PROGRAM Fast
VAR
	SerialLineControl1:SerialLineControl;
END_VAR

//编码器任务周期
serial1fast();

ACTION Serial1Fast:
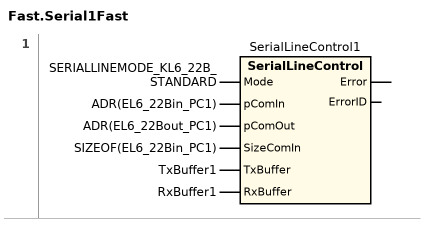
// NETWORK 1
SerialLineControl1(
    Mode := SERIALLINEMODE_KL6_22B_STANDARD,
    pComIn := ADR(EL6_22Bin_PC1),
    pComOut := ADR(EL6_22Bout_PC1),
    SizeComIn := SIZEOF(EL6_22Bin_PC1),
    TxBuffer := TxBuffer1,
    RxBuffer := RxBuffer1); // SerialLineControl
END_ACTION

END_PROGRAM

(* stored: Version 1.1.0.1, ProductVersion 3.1.0.38
   POU Fast: Id {5d8d0883-7042-4aab-b3e0-090e745570b4}, SpecialFunc None
   Action Serial1Fast: Id {6e45eeed-561d-45d2-992d-73bfbcd9c662} *)
